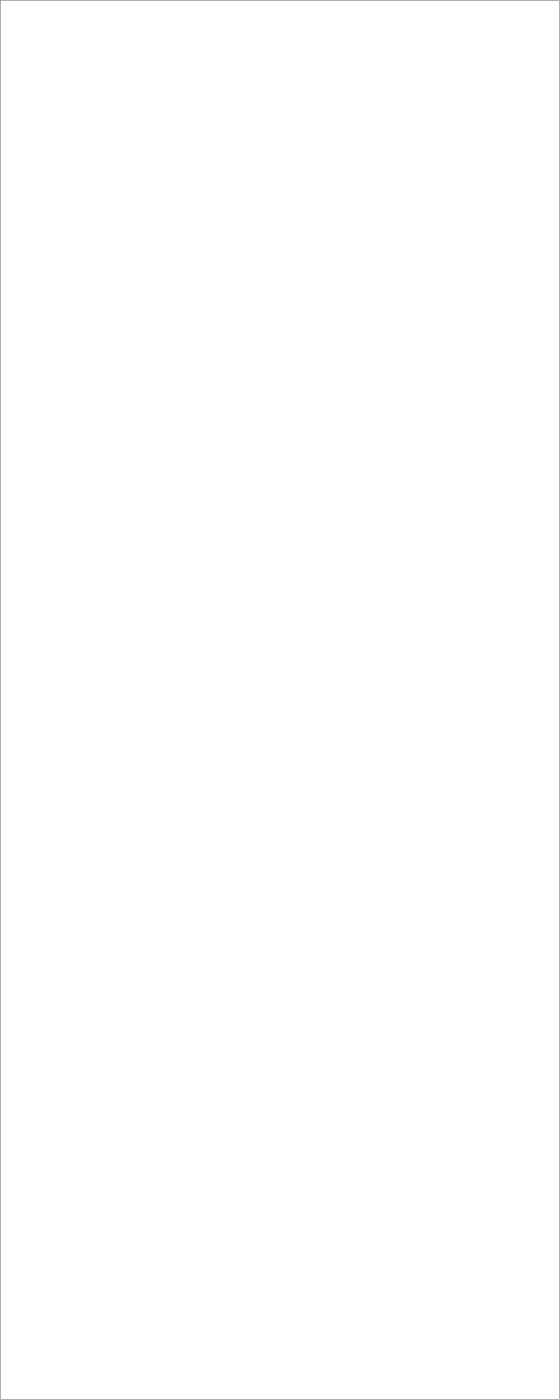
VISUALIZATION HMI_SenSimTest  // 801x2002
    Rectangle (7,175 430x823)
    Rectangle (260,175 176x823)
    Rectangle (7,875 429x23)
    Rectangle (7,741 429x23)
    Rectangle (7,174 429x23)
    Rectangle (6,16 669x143)
    Rectangle (6,17 669x32), "Manual Command Simulation From PLC"
    Checkbox (395,232 30x31), "Checkbox", tooltip "Enable Simulation", variable: stHMITIISenSimArray[iHMICbLevelSelection].bHMITIIByPassArray[1]
    ComboBoxInteger (295,235 100x25), tooltip "BackDoorSimulationMode", variable: arrTCMultiLevel[iHMICbLevelSelection].fbTCMultiLevelSeq.stMLBIO.ipAPPresentSensor, text list: 'BDList'
    RoundedRectangle (265,234 26x26), tooltip "VIO Status", colour toggle: arrTCMultiLevel[iHMICbLevelSelection].fbTCMultiLevelSeq.stMLVIO.ipAPPresentSensor
    Checkbox (263,201 164x31), "TIISen:VIOSim Override", variable: bHMIEnTIISenSimulation
    Checkbox (395,263 30x31), "Checkbox", tooltip "Enable Simulation", variable: stHMITIISenSimArray[iHMICbLevelSelection].bHMITIIByPassArray[2]
    ComboBoxInteger (295,267 100x25), tooltip "BackDoorSimulationMode", variable: arrTCMultiLevel[iHMICbLevelSelection].fbTCMultiLevelSeq.stMLBIO.ipAPPowerOn, text list: 'BDList'
    RoundedRectangle (265,265 26x26), tooltip "VIO Status", colour toggle: arrTCMultiLevel[iHMICbLevelSelection].fbTCMultiLevelSeq.stMLVIO.ipAPPowerOn
    Checkbox (395,294 30x31), "Checkbox", tooltip "Enable Simulation", variable: stHMITIISenSimArray[iHMICbLevelSelection].bHMITIIByPassArray[3]
    ComboBoxInteger (295,298 100x25), tooltip "BackDoorSimulationMode", variable: arrTCMultiLevel[iHMICbLevelSelection].fbTCMultiLevelSeq.stMLBIO.ipAPReady, text list: 'BDList'
    RoundedRectangle (265,296 26x26), tooltip "VIO Status", colour toggle: arrTCMultiLevel[iHMICbLevelSelection].fbTCMultiLevelSeq.stMLVIO.ipAPReady
    Checkbox (395,325 30x31), "Checkbox", tooltip "Enable Simulation", variable: stHMITIISenSimArray[iHMICbLevelSelection].bHMITIIByPassArray[4]
    ComboBoxInteger (295,328 100x25), tooltip "BackDoorSimulationMode", variable: arrTCMultiLevel[iHMICbLevelSelection].fbTCMultiLevelSeq.stMLBIO.ipHandlerSafeToEnterPLC, text list: 'BDList'
    RoundedRectangle (265,327 26x26), tooltip "VIO Status", colour toggle: arrTCMultiLevel[iHMICbLevelSelection].fbTCMultiLevelSeq.stMLVIO.ipHandlerSafeToEnterPLC
    Checkbox (395,356 30x31), "Checkbox", tooltip "Enable Simulation", variable: stHMITIISenSimArray[iHMICbLevelSelection].bHMITIIByPassArray[5]
    ComboBoxInteger (295,359 100x25), tooltip "BackDoorSimulationMode", variable: arrTCMultiLevel[iHMICbLevelSelection].fbTCMultiLevelSeq.stMLBIO.ipHandlerSafeToEnterHwr, text list: 'BDList'
    RoundedRectangle (265,358 26x26), tooltip "VIO Status", colour toggle: arrTCMultiLevel[iHMICbLevelSelection].fbTCMultiLevelSeq.stMLVIO.ipHandlerSafeToEnterHwr
    Checkbox (395,387 30x31), "Checkbox", tooltip "Enable Simulation", variable: stHMITIISenSimArray[iHMICbLevelSelection].bHMITIIByPassArray[6]
    ComboBoxInteger (295,390 100x25), tooltip "BackDoorSimulationMode", variable: arrTCMultiLevel[iHMICbLevelSelection].fbTCMultiLevelSeq.stMLBIO.ipCellFluidLeakage1, text list: 'BDList'
    RoundedRectangle (265,389 26x26), tooltip "VIO Status", colour toggle: arrTCMultiLevel[iHMICbLevelSelection].fbTCMultiLevelSeq.stMLVIO.ipCellFluidLeakage1
    Checkbox (395,418 30x31), "Checkbox", tooltip "Enable Simulation", variable: stHMITIISenSimArray[iHMICbLevelSelection].bHMITIIByPassArray[7]
    ComboBoxInteger (295,421 100x25), tooltip "BackDoorSimulationMode", variable: arrTCMultiLevel[iHMICbLevelSelection].fbTCMultiLevelSeq.stMLBIO.ipCellFluidLeakage2, text list: 'BDList'
    RoundedRectangle (265,420 26x26), tooltip "VIO Status", colour toggle: arrTCMultiLevel[iHMICbLevelSelection].fbTCMultiLevelSeq.stMLVIO.ipCellFluidLeakage2
    Checkbox (395,449 30x31), "Checkbox", tooltip "Enable Simulation", variable: stHMITIISenSimArray[iHMICbLevelSelection].bHMITIIByPassArray[8]
    ComboBoxInteger (295,452 100x25), tooltip "BackDoorSimulationMode", variable: arrTCMultiLevel[iHMICbLevelSelection].fbTCMultiLevelSeq.stMLBIO.ipCellGroundFault, text list: 'BDList'
    RoundedRectangle (265,451 26x26), tooltip "VIO Status", colour toggle: arrTCMultiLevel[iHMICbLevelSelection].fbTCMultiLevelSeq.stMLVIO.ipCellGroundFault
    Checkbox (395,480 30x31), "Checkbox", tooltip "Enable Simulation", variable: stHMITIISenSimArray[iHMICbLevelSelection].bHMITIIByPassArray[9]
    ComboBoxInteger (295,483 100x25), tooltip "BackDoorSimulationMode", variable: arrTCMultiLevel[iHMICbLevelSelection].fbTCMultiLevelSeq.stMLBIO.ipTesterPresent, text list: 'BDList'
    RoundedRectangle (265,482 26x26), tooltip "VIO Status", colour toggle: arrTCMultiLevel[iHMICbLevelSelection].fbTCMultiLevelSeq.stMLVIO.ipTesterPresent
    Checkbox (395,511 30x31), "Checkbox", tooltip "Enable Simulation", variable: stHMITIISenSimArray[iHMICbLevelSelection].bHMITIIByPassArray[10]
    ComboBoxInteger (295,514 100x25), tooltip "BackDoorSimulationMode", variable: arrTCMultiLevel[iHMICbLevelSelection].fbTCMultiLevelSeq.stMLBIO.ipTesterPowerOn, text list: 'BDList'
    RoundedRectangle (265,513 26x26), tooltip "VIO Status", colour toggle: arrTCMultiLevel[iHMICbLevelSelection].fbTCMultiLevelSeq.stMLVIO.ipTesterPowerOn
    Checkbox (395,542 30x31), "Checkbox", tooltip "Enable Simulation", variable: stHMITIISenSimArray[iHMICbLevelSelection].bHMITIIByPassArray[11]
    ComboBoxInteger (295,545 100x25), tooltip "BackDoorSimulationMode", variable: arrTCMultiLevel[iHMICbLevelSelection].fbTCMultiLevelSeq.stMLBIO.ipTesterReady, text list: 'BDList'
    RoundedRectangle (265,544 26x26), tooltip "VIO Status", colour toggle: arrTCMultiLevel[iHMICbLevelSelection].fbTCMultiLevelSeq.stMLVIO.ipTesterReady
    Checkbox (395,573 30x31), "Checkbox", tooltip "Enable Simulation", variable: stHMITIISenSimArray[iHMICbLevelSelection].bHMITIIByPassArray[12]
    ComboBoxInteger (295,576 100x25), tooltip "BackDoorSimulationMode", variable: arrTCMultiLevel[iHMICbLevelSelection].fbTCMultiLevelSeq.stMLBIO.ipTCCellDoorClosed, text list: 'BDList'
    RoundedRectangle (265,575 26x26), tooltip "VIO Status", colour toggle: arrTCMultiLevel[iHMICbLevelSelection].fbTCMultiLevelSeq.stMLVIO.ipTCCellDoorClosed
    Checkbox (395,604 30x31), "Checkbox", tooltip "Enable Simulation", variable: stHMITIISenSimArray[iHMICbLevelSelection].bHMITIIByPassArray[13]
    ComboBoxInteger (295,607 100x25), tooltip "BackDoorSimulationMode", variable: arrTCMultiLevel[iHMICbLevelSelection].fbTCMultiLevelSeq.stMLBIO.ipTesterLatchesClosed, text list: 'BDList'
    RoundedRectangle (265,606 26x26), tooltip "VIO Status", colour toggle: arrTCMultiLevel[iHMICbLevelSelection].fbTCMultiLevelSeq.stMLVIO.ipTesterLatchesClosed
    Checkbox (395,635 30x31), "Checkbox", tooltip "Enable Simulation", variable: stHMITIISenSimArray[iHMICbLevelSelection].bHMITIIByPassArray[14]
    ComboBoxInteger (295,638 100x25), tooltip "BackDoorSimulationMode", variable: arrTCMultiLevel[iHMICbLevelSelection].fbTCMultiLevelSeq.stMLBIO.ipTIUPresent, text list: 'BDList'
    RoundedRectangle (265,637 26x26), tooltip "VIO Status", colour toggle: arrTCMultiLevel[iHMICbLevelSelection].fbTCMultiLevelSeq.stMLVIO.ipTIUPresent
    Checkbox (395,666 30x31), "Checkbox", tooltip "Enable Simulation"
    ComboBoxInteger (295,669 100x25), tooltip "BackDoorSimulationMode", variable: arrTCMultiLevel[iHMICbLevelSelection].fbTCMultiLevelSeq.stMLBIO.ipAPPresentSensor, text list: 'BDList'
    RoundedRectangle (265,668 26x26), tooltip "VIO Status"
    Checkbox (395,697 30x31), "Checkbox", tooltip "Enable Simulation"
    ComboBoxInteger (295,700 100x25), tooltip "BackDoorSimulationMode", variable: arrTCMultiLevel[iHMICbLevelSelection].fbTCMultiLevelSeq.stMLBIO.ipAPPresentSensor, text list: 'BDList'
    RoundedRectangle (265,699 26x26), tooltip "VIO Status"
    RoundedRectangle (69,234 165x25), "01)_AP_PresentSensor*"
    Checkbox (12,232 30x31), "Checkbox", tooltip "Enable Simulation", variable: stHMITIIByPassArray[iHMICbLevelSelection].bHMITIIByPassArray[1]
    RoundedRectangle (69,265 165x25), "02)_AP_PowerOn*"
    Checkbox (12,263 30x31), "Checkbox", tooltip "Enable Simulation", variable: stHMITIIByPassArray[iHMICbLevelSelection].bHMITIIByPassArray[2]
    RoundedRectangle (69,296 165x25), "03)_AP_Ready"
    Checkbox (12,294 30x31), "Checkbox", tooltip "Enable Simulation", variable: stHMITIIByPassArray[iHMICbLevelSelection].bHMITIIByPassArray[3]
    RoundedRectangle (69,327 165x25), "04)_AP_DeactuatedPLC`*`"
    Checkbox (12,325 30x31), "Checkbox", tooltip "Enable Simulation", variable: stHMITIIByPassArray[iHMICbLevelSelection].bHMITIIByPassArray[4]
    RoundedRectangle (69,358 165x25), "05)_AP_DeactuatedHwr`*`"
    Checkbox (12,356 30x31), "Checkbox", tooltip "Enable Simulation", variable: stHMITIIByPassArray[iHMICbLevelSelection].bHMITIIByPassArray[5]
    RoundedRectangle (69,389 165x25), "06)_CellFluidLeakage1"
    Checkbox (12,387 30x31), "Checkbox", tooltip "Enable Simulation", variable: stHMITIIByPassArray[iHMICbLevelSelection].bHMITIIByPassArray[6]
    RoundedRectangle (69,420 165x25), "07)_CellFluidLeakage2"
    Checkbox (12,418 30x31), "Checkbox", tooltip "Enable Simulation", variable: stHMITIIByPassArray[iHMICbLevelSelection].bHMITIIByPassArray[7]
    RoundedRectangle (69,451 165x25), "08)_CellGroundFault"
    Checkbox (12,449 30x31), "Checkbox", tooltip "Enable Simulation", variable: stHMITIIByPassArray[iHMICbLevelSelection].bHMITIIByPassArray[8]
    RoundedRectangle (69,482 165x25), "09)_TesterPresent**"
    Checkbox (12,480 30x31), "Checkbox", tooltip "Enable Simulation", variable: stHMITIIByPassArray[iHMICbLevelSelection].bHMITIIByPassArray[9]
    RoundedRectangle (69,513 165x25), "10)_TesterPowerOn**"
    Checkbox (12,511 30x31), "Checkbox", tooltip "Enable Simulation", variable: stHMITIIByPassArray[iHMICbLevelSelection].bHMITIIByPassArray[10]
    RoundedRectangle (69,544 165x25), "11)_TesterReady"
    Checkbox (12,542 30x31), "Checkbox", tooltip "Enable Simulation", variable: stHMITIIByPassArray[iHMICbLevelSelection].bHMITIIByPassArray[11]
    RoundedRectangle (69,575 165x25), "12)_TCCellDoorClosed"
    Checkbox (12,573 30x31), "Checkbox", tooltip "Enable Simulation", variable: stHMITIIByPassArray[iHMICbLevelSelection].bHMITIIByPassArray[12]
    RoundedRectangle (69,606 165x25), "13)_TesterLatchesClosed**"
    Checkbox (12,604 30x31), "Checkbox", tooltip "Enable Simulation", variable: stHMITIIByPassArray[iHMICbLevelSelection].bHMITIIByPassArray[13]
    RoundedRectangle (69,637 165x25), "14)_TIUPresent"
    Checkbox (12,635 30x31), "Checkbox", tooltip "Enable Simulation", variable: stHMITIIByPassArray[iHMICbLevelSelection].bHMITIIByPassArray[14]
    RoundedRectangle (69,668 165x25)
    Checkbox (12,666 30x31), "Checkbox", tooltip "Enable Simulation"
    RoundedRectangle (69,699 165x25)
    Checkbox (12,697 30x31), "Checkbox", tooltip "Enable Simulation"
    Checkbox (12,202 227x31), "TII Alarm Enable Override", variable: bHMITIIBypass
    Checkbox (629,331 30x31), "Checkbox", tooltip "Enable Simulation", variable: stHMIBtnSimArray[iHMICbLevelSelection].bHMITIIByPassArray[1]
    ComboBoxInteger (483,334 140x25), tooltip "BackDoorSimulationMode", variable: arrTCMultiLevel[iHMICbLevelSelection].fbTCMultiLevelSeq.stMLBIO.ipDrawerMaintenanceModeBtn, text list: 'BDList'
    RoundedRectangle (453,333 26x26), tooltip "VIO Status", colour toggle: arrTCMultiLevel[iHMICbLevelSelection].fbTCMultiLevelSeq.stMLVIO.ipDrawerMaintenanceModeBtn
    Checkbox (629,362 30x31), "Checkbox", tooltip "Enable Simulation", variable: stHMIBtnSimArray[iHMICbLevelSelection].bHMITIIByPassArray[2]
    ComboBoxInteger (483,366 140x25), tooltip "BackDoorSimulationMode", variable: arrTCMultiLevel[iHMICbLevelSelection].fbTCMultiLevelSeq.stMLBIO.ipTCCellAbortFlowBtn, text list: 'BDList'
    RoundedRectangle (453,364 26x26), tooltip "VIO Status", colour toggle: arrTCMultiLevel[iHMICbLevelSelection].fbTCMultiLevelSeq.stMLVIO.ipTCCellAbortFlowBtn
    Checkbox (629,393 30x31), "Checkbox", tooltip "Enable Simulation", variable: stHMIBtnSimArray[iHMICbLevelSelection].bHMITIIByPassArray[3]
    ComboBoxInteger (483,397 140x25), tooltip "BackDoorSimulationMode", variable: arrTCMultiLevel[iHMICbLevelSelection].fbTCMultiLevelSeq.stMLBIO.ipTCCellDoorOpenReqBtn, text list: 'BDList'
    RoundedRectangle (453,395 26x26), tooltip "VIO Status", colour toggle: arrTCMultiLevel[iHMICbLevelSelection].fbTCMultiLevelSeq.stMLVIO.ipTCCellDoorOpenReqBtn
    Checkbox (452,300 157x31), "Btn VIO Sim Override", variable: bHMIBtnSimulation
    Checkbox (454,427 150x30), "AutoRsetEvntTrigger", variable: bHMIRsetEvntTriggerOnProductionMode
    RoundedRectangle (41,234 26x26), tooltip "VIO Status", colour toggle: ALMTC.Level[iHMICbLevelSelection].AlarmID[1]
    RoundedRectangle (41,265 26x26), tooltip "VIO Status", colour toggle: ALMTC.Level[iHMICbLevelSelection].AlarmID[2]
    RoundedRectangle (41,296 26x26), tooltip "VIO Status", colour toggle: ALMTC.Level[iHMICbLevelSelection].AlarmID[3]
    RoundedRectangle (41,327 26x26), tooltip "VIO Status", colour toggle: ALMTC.Level[iHMICbLevelSelection].AlarmID[4]
    RoundedRectangle (41,358 26x26), tooltip "VIO Status", colour toggle: ALMTC.Level[iHMICbLevelSelection].AlarmID[5]
    RoundedRectangle (41,389 26x26), tooltip "VIO Status", colour toggle: ALMTC.Level[iHMICbLevelSelection].AlarmID[6]
    RoundedRectangle (41,420 26x26), tooltip "VIO Status", colour toggle: ALMTC.Level[iHMICbLevelSelection].AlarmID[7]
    RoundedRectangle (41,451 26x26), tooltip "VIO Status", colour toggle: ALMTC.Level[iHMICbLevelSelection].AlarmID[8]
    RoundedRectangle (41,482 26x26), tooltip "VIO Status", colour toggle: ALMTC.Level[iHMICbLevelSelection].AlarmID[9]
    RoundedRectangle (41,513 26x26), tooltip "VIO Status", colour toggle: ALMTC.Level[iHMICbLevelSelection].AlarmID[10]
    RoundedRectangle (41,544 26x26), tooltip "VIO Status", colour toggle: ALMTC.Level[iHMICbLevelSelection].AlarmID[11]
    RoundedRectangle (41,575 26x26), tooltip "VIO Status", colour toggle: ALMTC.Level[iHMICbLevelSelection].AlarmID[12]
    RoundedRectangle (41,606 26x26), tooltip "VIO Status", colour toggle: ALMTC.Level[iHMICbLevelSelection].AlarmID[13]
    RoundedRectangle (41,637 26x26), tooltip "VIO Status", colour toggle: ALMTC.Level[iHMICbLevelSelection].AlarmID[14]
    RoundedRectangle (41,668 26x26), tooltip "VIO Status"
    RoundedRectangle (41,699 26x26), tooltip "VIO Status"
    Checkbox (394,766 30x31), "Checkbox", tooltip "Enable Simulation", variable: bHMIColSenSimArray[1]
    ComboBoxInteger (294,769 100x25), tooltip "BackDoorSimulationMode", variable: fbTCColumn.stTCColumnBIO.ipColumnFluid_PCW_Leakage, text list: 'BDList'
    RoundedRectangle (264,768 26x26), tooltip "VIO Status", colour toggle: fbTCColumn.stTCColumnVIO.ipColumnFluid_PCW_Leakage
    Checkbox (394,797 30x31), "Checkbox", tooltip "Enable Simulation", variable: bHMIColSenSimArray[2]
    ComboBoxInteger (294,800 100x25), tooltip "BackDoorSimulationMode", variable: fbTCColumn.stTCColumnBIO.ipAllTCDrawerRetractedinCell, text list: 'BDList'
    RoundedRectangle (264,799 26x26), tooltip "VIO Status", colour toggle: fbTCColumn.stTCColumnVIO.ipAllTCDrawerRetractedinCell
    Checkbox (394,828 30x31), "Checkbox", tooltip "Enable Simulation", variable: bHMIColSenSimArray[3]
    ComboBoxInteger (294,831 100x25), tooltip "BackDoorSimulationMode", variable: fbTCColumn.stTCColumnBIO.ipSystem_ipColumnGroundFault, text list: 'BDList'
    RoundedRectangle (264,830 26x26), tooltip "VIO Status", colour toggle: fbTCColumn.stTCColumnVIO.ipSystem_ipColumnGroundFault
    RoundedRectangle (71,769 162x25), "1)_Col_Leakage"
    Checkbox (12,767 30x31), "Checkbox", tooltip "Enable Simulation", variable: arrHMISysAlmByPass[1]
    RoundedRectangle (71,800 162x25), "2)_All_Dwr_Ret"
    Checkbox (12,799 30x31), "Checkbox", tooltip "Enable Simulation", variable: arrHMISysAlmByPass[2]
    RoundedRectangle (71,831 162x25), "3)_Col_Grd"
    Checkbox (12,830 30x31), "Checkbox", tooltip "Enable Simulation", variable: arrHMISysAlmByPass[3]
    RoundedRectangle (42,769 26x26), tooltip "VIO Status", colour toggle: ALMTC.Common.AlarmID[1]
    RoundedRectangle (42,800 26x26), tooltip "VIO Status", colour toggle: ALMTC.Common.AlarmID[2]
    RoundedRectangle (42,831 26x26), tooltip "VIO Status", colour toggle: ALMTC.Common.AlarmID[3]
    RoundedRectangle (476,233 181x25), "ButtonModeConditionSimulation"
        toggle arrHMIBtnSolidOn_Condition[iHMICbLevelSelection,iHMIBtnType]
    RoundedRectangle (449,233 25x25), colour toggle: arrHMIBtnSolidOn_Condition[iHMICbLevelSelection,iHMIBtnType]
    ComboBoxInteger (451,266 208x25), tooltip "BackDoorSimulationMode", variable: iHMIBtnType, text list: 'BtnTxtList'
    ComboBoxInteger (106,71 188x30), variable: iHMICbCmdSelection, text list: 'CmdTxtList'
    ComboBoxInteger (14,71 89x30), variable: iHMICbLevelSelection, text list: 'LevelTxtList'
    Button (12,108 281x45), "Test Command"
        tap TestManually.bTestCommand
    ComboBoxInteger (306,73 276x25), variable: TestManually.iAlarmCode, text list: 'AlarmTxtList'
    Checkbox (586,68 37x30), variable: bHMIResetAllAlarm
    Label (616,68 183x30), "Reset All"
    Label (304,50 215x30), "Individual Alarm ID:"
    Button (302,111 281x42), "Init All Level"
        tap TestManually.bInitialiseAll
    Checkbox (397,900 30x31), "Checkbox", tooltip "Enable Simulation", variable: stDebugStation.fbDBStnSeq.bTIISenSimArray[1]
    ComboBoxInteger (297,903 100x25), tooltip "BackDoorSimulationMode", variable: stDebugStation.fbDBStnSeq.stDebugStationBIO.ipDBStnAPPresentSensor, text list: 'BDList'
    RoundedRectangle (267,902 26x26), tooltip "VIO Status", colour toggle: stDebugStation.fbDBStnSeq.stDebugStationVIO.ipDBStnAPPresentSensor
    Checkbox (397,931 30x31), "Checkbox", tooltip "Enable Simulation", variable: stDebugStation.fbDBStnSeq.bTIISenSimArray[2]
    ComboBoxInteger (297,935 100x25), tooltip "BackDoorSimulationMode", variable: stDebugStation.fbDBStnSeq.stDebugStationBIO.ipDBStnAPPowerOn, text list: 'BDList'
    RoundedRectangle (267,933 26x26), tooltip "VIO Status", colour toggle: stDebugStation.fbDBStnSeq.stDebugStationVIO.ipDBStnAPPowerOn
    Checkbox (397,962 30x31), "Checkbox", tooltip "Enable Simulation", variable: stDebugStation.fbDBStnSeq.bTIISenSimArray[3]
    ComboBoxInteger (297,966 100x25), tooltip "BackDoorSimulationMode", variable: stDebugStation.fbDBStnSeq.stDebugStationBIO.ipDBStnAPReady, text list: 'BDList'
    RoundedRectangle (267,964 26x26), tooltip "VIO Status", colour toggle: stDebugStation.fbDBStnSeq.stDebugStationVIO.ipDBStnAPReady
    RoundedRectangle (71,902 165x25), "01)_AP_PresentSensor"
    Checkbox (14,900 30x31), "Checkbox", tooltip "Enable Simulation", variable: stHMITIIByPassArray[iHMICbLevelSelection].bHMITIIByPassArray[1]
    RoundedRectangle (71,933 165x25), "02)_AP_PowerOn"
    Checkbox (14,931 30x31), "Checkbox", tooltip "Enable Simulation", variable: stHMITIIByPassArray[iHMICbLevelSelection].bHMITIIByPassArray[2]
    RoundedRectangle (71,964 165x25), "03)_AP_Ready"
    Checkbox (14,962 30x31), "Checkbox", tooltip "Enable Simulation", variable: stHMITIIByPassArray[iHMICbLevelSelection].bHMITIIByPassArray[3]
    RoundedRectangle (43,902 26x26), tooltip "VIO Status", colour toggle: ALMTC.Level[iHMICbLevelSelection].AlarmID[1]
    RoundedRectangle (43,933 26x26), tooltip "VIO Status", colour toggle: ALMTC.Level[iHMICbLevelSelection].AlarmID[2]
    RoundedRectangle (43,964 26x26), tooltip "VIO Status", colour toggle: ALMTC.Level[iHMICbLevelSelection].AlarmID[3]
    Label (20,871 183x30), "DEBUG STATION"
    Label (15,171 183x30), "CELL STACK"
    Label (20,740 183x30), "COLUMN"
    Group (452,468 225x262)
        Rectangle (0,0 215x259)
        Rectangle (0,237 215x22)
        RoundedRectangle (7,206 60x26), "Level[1]", tooltip "VIO Status", colour toggle: TC_ModuleState[1].Tester = E_State.eEnabled
        RoundedRectangle (7,177 60x26), "Level[2]", tooltip "VIO Status", colour toggle: TC_ModuleState[2].Tester= E_State.eEnabled
        RoundedRectangle (7,148 60x26), "Level[3]", tooltip "VIO Status", colour toggle: TC_ModuleState[3].Tester = E_State.eEnabled
        RoundedRectangle (7,119 60x26), "Level[4]", tooltip "VIO Status", colour toggle: TC_ModuleState[4].Tester = E_State.eEnabled
        RoundedRectangle (7,90 60x26), "Level[5]", tooltip "VIO Status", colour toggle: TC_ModuleState[5].Tester = E_State.eEnabled
        RoundedRectangle (7,61 60x26), "Level[6]", tooltip "VIO Status", colour toggle: TC_ModuleState[6].Tester = E_State.eEnabled
        Label (6,32 61x30), "Tester"
        RoundedRectangle (149,206 60x26), "Level[1]", tooltip "VIO Status", colour toggle: TC_ModuleState[1].TCSite[1].TIERII = E_State.eEnabled
        RoundedRectangle (149,177 60x26), "Level[2]", tooltip "VIO Status", colour toggle: TC_ModuleState[2].TCSite[1].TIERII = E_State.eEnabled
        RoundedRectangle (149,148 60x26), "Level[3]", tooltip "VIO Status", colour toggle: TC_ModuleState[3].TCSite[1].TIERII = E_State.eEnabled
        RoundedRectangle (149,119 60x26), "Level[4]", tooltip "VIO Status", colour toggle: TC_ModuleState[4].TCSite[1].TIERII = E_State.eEnabled
        RoundedRectangle (149,90 60x26), "Level[5]", tooltip "VIO Status", colour toggle: TC_ModuleState[5].TCSite[1].TIERII = E_State.eEnabled
        RoundedRectangle (149,61 60x26), "Level[6]", tooltip "VIO Status", colour toggle: TC_ModuleState[6].TCSite[1].TIERII = E_State.eEnabled
        Label (162,32 32x30), "TII"
        RoundedRectangle (78,207 60x26), "Level[1]", tooltip "VIO Status", colour toggle: TC_ModuleState[1].TCSite[1].TCU = E_State.eEnabled
        RoundedRectangle (78,178 60x26), "Level[2]", tooltip "VIO Status", colour toggle: TC_ModuleState[2].TCSite[1].TCU= E_State.eEnabled
        RoundedRectangle (78,149 60x26), "Level[3]", tooltip "VIO Status", colour toggle: TC_ModuleState[3].TCSite[1].TCU = E_State.eEnabled
        RoundedRectangle (78,120 60x26), "Level[4]", tooltip "VIO Status", colour toggle: TC_ModuleState[4].TCSite[1].TCU = E_State.eEnabled
        RoundedRectangle (78,91 60x26), "Level[5]", tooltip "VIO Status", colour toggle: TC_ModuleState[5].TCSite[1].TCU = E_State.eEnabled
        RoundedRectangle (78,62 60x26), "Level[6]", tooltip "VIO Status", colour toggle: TC_ModuleState[6].TCSite[1].TCU = E_State.eEnabled
        Label (87,33 43x30), "TCU"
        Label (12,232 213x30), "Green: Enable , Gray: Disable"
        Rectangle (0,1 215x32), "Enable/ Disable Status"
    Rectangle (7,1009 430x271)
    Rectangle (7,1010 429x32), "Manual Command Simulation From PLC"
    Label (9,1073 153x30), "AP240PwrCheckDelay(ms)"
    Textfield (162,1073 103x30), "%i", text variable: APPwrOnChkDelay, input disabled if: TRUE
        OnMouseClick: write the text variable via Default
    Button (383,1074 50x30), "Write", input disabled if: NOT (iAPPwrOnChkDelay>=0)
        tap BtnSetAPPwrOnChkDelay
    Label (165,1047 78x30), "Current Value"
    Label (276,1046 84x30), "Value To Write"
    Textfield (272,1073 103x30), "%i", text variable: iAPPwrOnChkDelay
        OnMouseClick: write the text variable via Default
    Label (8,1109 154x30), "Tst240PwrCheckDelay(ms)"
    Textfield (162,1109 103x30), "%i", text variable: TstPwrOnChkDelay, input disabled if: TRUE
        OnMouseClick: write the text variable via Default
    Button (383,1110 50x30), "Write", input disabled if: NOT (iTstPwrOnChkDelay>=0)
        tap BtnSetTstPwrOnChkDelay
    Textfield (272,1109 103x30), "%i", text variable: iTstPwrOnChkDelay
        OnMouseClick: write the text variable via Default
    Label (9,1150 153x30), "APReadyCheckDelay(ms)"
    Textfield (162,1150 103x30), "%i", text variable: APPwrOnChkDelay, input disabled if: TRUE
        OnMouseClick: write the text variable via Default
    Button (383,1151 50x30), "Write", input disabled if: NOT (iAPPwrOnChkDelay>=0)
        tap BtnSetAPPwrOnChkDelay
    Textfield (272,1150 103x30), "%i", text variable: iAPPwrOnChkDelay
        OnMouseClick: write the text variable via Default
    Label (8,1186 154x30), "TstReadyCheckDelay(ms)"
    Textfield (162,1186 103x30), "%i", text variable: TstPwrOnChkDelay, input disabled if: TRUE
        OnMouseClick: write the text variable via Default
    Button (383,1187 50x30), "Write", input disabled if: NOT (iTstPwrOnChkDelay>=0)
        tap BtnSetTstPwrOnChkDelay
    Textfield (272,1186 103x30), "%i", text variable: iTstPwrOnChkDelay
        OnMouseClick: write the text variable via Default
    Rectangle (0,0 792x2000), invisible if: bEnableManualCommandTest1 AND bEnableManualCommandTest2
END_VISUALIZATION

(* stored: Version 1.1.0.1, ProductVersion 3.1.4022.12
   Visu HMI_SenSimTest: Id {935d0c8b-5a4a-4123-bec5-8e0ae35adbc3} *)
